PROGRAM branch
VAR
END_VAR

END_PROGRAM

(* stored: Version 1.1.0.1, ProductVersion 3.1.4024.12
   POU branch: Id {75db8dd7-c841-0d3e-204f-78e5e354675e}, SpecialFunc None *)
